FUNCTION_BLOCK Test_StringToIpAddress EXTENDS T_UnitTestBase
VAR_INPUT
END_VAR
VAR_OUTPUT
END_VAR
VAR
	SubjectString : T_MaxString := '192.168.1.120';
	Result : ARRAY[1..4] OF BYTE;
END_VAR

Result := F_String_To_IPv4_Address(SubjectString);

Assertion.AssertEquals_BYTE(
	Expected := 120,
	Actual := Result[1],
	VariableName := 'F_String_To_IPv4_Address(SubjectString)');
	
Assertion.AssertEquals_BYTE(
	Expected := 1,
	Actual := Result[2],
	VariableName := 'F_String_To_IPv4_Address(SubjectString)');
	
Assertion.AssertEquals_BYTE(
	Expected := 168,
	Actual := Result[3],
	VariableName := 'F_String_To_IPv4_Address(SubjectString)');
	
Assertion.AssertEquals_BYTE(
	Expected := 192,
	Actual := Result[4],
	VariableName := 'F_String_To_IPv4_Address(SubjectString)');
	
TestFinished();

END_FUNCTION_BLOCK

(* stored: Version 1.1.0.1, ProductVersion 3.1.4024.9
   POU Test_StringToIpAddress: Id {5bc33b48-a377-05a1-2065-47bed9f2c7ae}, SpecialFunc None *)
